{attribute 'qualified_only'}
VAR_GLOBAL
		EC1 : EC1_DFE7C435;
END_VAR

(* stored: Version 1.2.0.0
   GVL GVL_iXlinker: Id {b555b60c-e215-4bfc-aaff-03687217c4e8} *)
